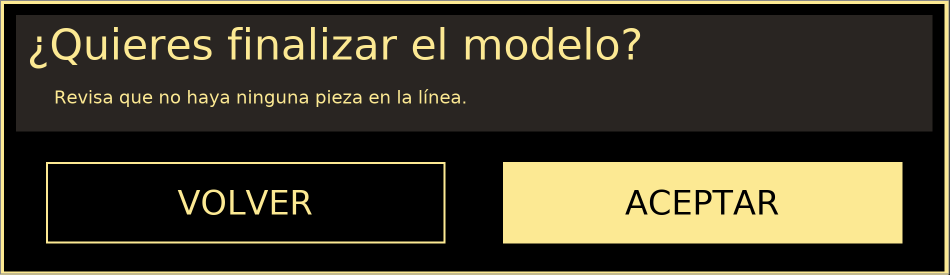
VISUALIZATION V_Emerg_Fin_Prod_Ch3  // 950x275
    Rectangle (0,0 948x275)
    Rectangle (16,15 916x116)
    Label (24,17 898x65), "¿Quieres finalizar el modelo?"
    Label (51,85 857x43), "Revisa que no haya ninguna pieza en la línea."
    Rectangle (503,162 399x81), "ACEPTAR"
        tap FuncParoNodoLocalCorteH3.FunGeneCortHum3.P_FinProduccion
        OnMouseClick: CloseDialog Dialog=V_Emerg_Fin_Prod_Ch3, Result=None, NumpadKeypadSet=True
        OnMouseClick: OpenDialog Dialog=Modelo_Tabla_Ch3, OpenModal=True, OpenCentered=True
    Rectangle (46,162 399x81), "VOLVER"
        OnMouseClick: CloseDialog Dialog=V_Emerg_Fin_Prod_Ch2, Result=Cancel, NumpadKeypadSet=True
END_VISUALIZATION

(* stored: Version 1.1.0.1, ProductVersion 3.1.4024.12
   Visu V_Emerg_Fin_Prod_Ch3: Id {7451803c-12fa-47e9-a9a7-753a334376c9} *)
